Yaskawa INFORM job: X2_7,2(150,-90).JBI

/JOB
//NAME X2_7,2(150,-90)
//POS
///NPOS 31,31,31,3,0,0
///TOOL 0
///POSTYPE PULSE
///PULSE
C00000=-1903,-101039,-123464,-18,98414,30
C00001=37629,-83041,-126142,12125,101236,-40991
C00002=120710,-114236,-128002,-161,94425,-119
C00003=120626,-97263,-85517,-147,77002,-126
C00004=120624,-90603,-79512,-147,76729,-126
C00005=120619,-87609,-75876,-147,76029,-126
C00006=120612,-86998,-74157,-145,75286,-128
C00007=120630,-84931,-74575,-148,76604,-124
C00008=120635,-82574,-72610,-148,76606,-123
C00009=120636,-81941,-72345,-149,76768,-122
C00010=120635,-82574,-72610,-148,76606,-123
C00011=120623,-96358,-82912,-147,75863,-125
C00012=120643,-96591,-84648,-150,76812,-120
C00013=120640,-89962,-78640,-150,76521,-120
C00014=120640,-87399,-76229,-150,76354,-120
C00015=120632,-86713,-74265,-149,75498,-122
C00016=120630,-86551,-75442,-148,76306,-123
C00017=120611,-84912,-73908,-144,76204,-130
C00018=120616,-83150,-73182,-145,76663,-128
C00019=120611,-84912,-73908,-144,76204,-130
C00020=120607,-95796,-83038,-144,76230,-131
C00021=120623,-87424,-78135,-4974,77554,1131
C00022=120623,-86585,-74968,-5002,76042,1192
C00023=120623,-87260,-75250,-5004,75869,1199
C00024=120623,-87371,-75295,-5004,75876,1199
C00025=120621,-87568,-75289,-5005,75773,1205
C00026=120621,-87481,-75230,-5007,75741,1203
C00027=120623,-86357,-74872,-5001,76100,1190
C00028=120623,-87221,-78171,-4972,77680,1126
C00029=120710,-114236,-128002,-161,94425,-119
C00030=-1903,-101039,-123464,-18,98414,30
BC00000=178010,519809,1070018
BC00001=191681,449862,974626
BC00002=183494,409566,1070018
BC00003=183494,402220,1070018
BC00004=183494,402220,1070018
BC00005=183494,402220,1070018
BC00006=183494,402220,1070018
BC00007=183494,402220,1070018
BC00008=183494,402220,1070018
BC00009=183494,402220,1070018
BC00010=183494,402220,1070018
BC00011=183494,402220,1070018
BC00012=246532,400736,1069536
BC00013=246532,400736,1069536
BC00014=246532,400736,1069536
BC00015=246532,400736,1069536
BC00016=246532,400736,1069536
BC00017=246532,400736,1069536
BC00018=246532,400736,1069536
BC00019=246532,400736,1069536
BC00020=246532,400736,1069536
BC00021=173106,403917,1075139
BC00022=173805,399378,1071655
BC00023=174085,397563,1063031
BC00024=178863,397480,1063167
BC00025=232858,397286,1063829
BC00026=237637,397335,1063811
BC00027=237357,399151,1072434
BC00028=236657,403689,1075139
BC00029=183494,409566,1070018
BC00030=178010,519809,1070018
EC00000=-1330261,372643
EC00001=-1330261,372641
EC00002=-1330261,372643
EC00003=-1330261,372643
EC00004=-1330261,372643
EC00005=-1330261,372643
EC00006=-1330261,372643
EC00007=-1330261,372643
EC00008=-1330261,372643
EC00009=-1330261,372643
EC00010=-1330261,372643
EC00011=-1330261,372643
EC00012=-1330261,372643
EC00013=-1330261,372643
EC00014=-1330261,372643
EC00015=-1330261,372643
EC00016=-1330261,372643
EC00017=-1330261,372643
EC00018=-1330261,372643
EC00019=-1330261,372643
EC00020=-1330261,372643
EC00021=-1330261,372643
EC00022=-1330261,372643
EC00023=-1330261,372643
EC00024=-1330261,372643
EC00025=-1330261,372643
EC00026=-1330261,372643
EC00027=-1330261,372643
EC00028=-1330261,372643
EC00029=-1330261,372643
EC00030=-1330261,372643
///POSTYPE BASE
///RECTAN
///RCONF 0,0,0,0,1,0,0,0,0,0,0,0,0,0,0,0,0,0,0,0,0,0,0,0
P00006=2.006,1.622,-0.565,0.0000,0.0000,0.0000
P00021=0.073,2.058,-0.109,0.0000,0.0000,0.0000
P00022=2.006,1.622,-0.565,0.0000,0.0000,0.0000
//INST
///DATE 2024/04/06 15:25
///ATTR SC,RW
///GROUP1 RB1,BS1
///GROUP2 ST1
NOP
'X2_7,2(150,-90)
MOVJ C00000 BC00000 VJ=100.00  +MOVJ EC00000 VJ=100.00
CALL JOB:CLEAN-R1_KM_NEW
MOVJ C00001 BC00001 VJ=100.00  +MOVJ EC00001 VJ=100.00
MOVJ C00002 BC00002 VJ=100.00  +MOVJ EC00002 VJ=100.00
'Path S3593
SFTOF3D
MOVJ C00003 BC00003 VJ=100.00  +MOVJ EC00003 VJ=100.00
MOVL C00004 BC00004 V=666.7  +MOVJ EC00004 VJ=100.00
SMOVL C00005 BC00005 V=166.7  +MOVJ EC00005
SREFP 3 C00006 BC00006  +REFP EC00006
CALL JOB:SEARCH-R1-S13D
SET P021 P006
SFTON3D P021
SMOVL C00007 BC00007 V=250.0  +MOVJ EC00007
SMOVL C00008 BC00008 V=166.7  +MOVJ EC00008
SREFP 3 C00009 BC00009  +REFP EC00009
CALL JOB:SEARCH-R1-S13D
SET P021 P006
SFTON3D P021
SMOVL C00010 BC00010 V=250.0  +MOVJ EC00010
MOVL C00011 BC00011 V=1000.0  +MOVJ EC00011 VJ=100.00
'EndPath S3593
'Path S4333
SFTOF3D
MOVJ C00012 BC00012 VJ=100.00  +MOVJ EC00012 VJ=100.00
MOVL C00013 BC00013 V=666.7  +MOVJ EC00013 VJ=100.00
SMOVL C00014 BC00014 V=166.7  +MOVJ EC00014
SREFP 3 C00015 BC00015  +REFP EC00015
CALL JOB:SEARCH-R1-S13D
SET P022 P006
SFTON3D P022
SMOVL C00016 BC00016 V=250.0  +MOVJ EC00016
SMOVL C00017 BC00017 V=166.7  +MOVJ EC00017
SREFP 3 C00018 BC00018  +REFP EC00018
CALL JOB:SEARCH-R1-S13D
SET P022 P006
SFTON3D P022
SMOVL C00019 BC00019 V=250.0  +MOVJ EC00019
MOVL C00020 BC00020 V=1000.0  +MOVJ EC00020 VJ=100.00
'EndPath S4333
'Path W3596
SFTOF3D
SFTON3D P021
MOVJ C00021 BC00021 VJ=100.00  +MOVJ EC00021 VJ=100.00
SMOVL C00022 BC00022 V=666.7  +MOVJ EC00022
SMOVL C00023 BC00023 V=166.7 PL=0  +MOVJ EC00023
MACRO1 MJ#(0) ARGF21
ARCON
SMOVL C00024 BC00024 V=9.2  +MOVJ EC00024
SMOVL C00025 BC00025 V=9.2  +MOVJ EC00025
SMOVL C00026 BC00026 V=9.2  +MOVJ EC00026
ARCOF
SMOVL C00027 BC00027 V=800.0  +MOVJ EC00027
SMOVL C00028 BC00028 V=1000.0  +MOVJ EC00028
SFTOF3D
'EndPath W3596
MOVJ C00029 BC00029 VJ=100.00  +MOVJ EC00029 VJ=100.00
MOVJ C00030 BC00030 VJ=100.00  +MOVJ EC00030 VJ=100.00
END
